(* Schneider Machine Expert - Basic project XNOR Gate, file version 2.9.0.0 *)
(* ProjectInformations: Name=New project *)

HARDWARE
  Cpu 0: TM221C24R
  EthernetConfiguration: NetworkName=M221, IpAllocationMode=FixedAddress, IpAddress=0.0.0.0, SubnetMask=0.0.0.0
  SerialLineConfiguration: Baud=Baud19200, Parity=ParityEven, DataBits=DataBits8, StopBits=StopBits1, PhysicalMedium=PhysicalMediumRs485, SlaveId=1, Addressing=SlaveAddressing
  MastTask: UsePeriodScanMode=false, PeriodScan=100
  FastTask: Period=255
  CpuBehavior: StartingMode=StartAsPreviousState, AutoSaveRamOnEeprom=true, WatchdogPeriod=250

SYMBOLS  (address, symbol, comment, settings)
  %I0.0     SWITCH_1
  %I0.1     SWITCH_2
  %Q0.0     MOTOR

POU New POU
  (* SectionNumber=1 *)

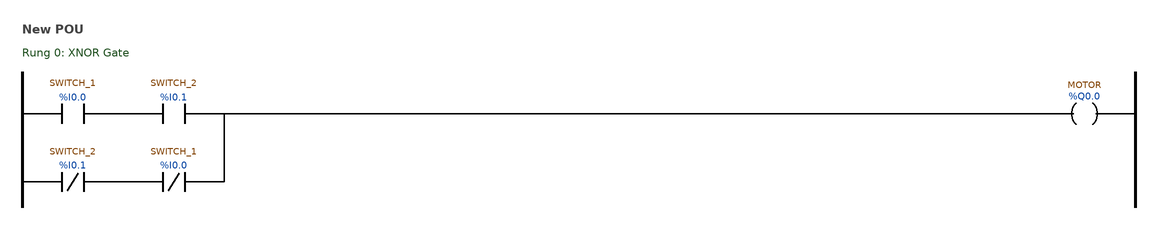

// Rung 0: XNOR Gate
  LD %I0.0                (* SWITCH_1 *)
  AND %I0.1               (* SWITCH_2 *)
  OR(N %I0.1              (* SWITCH_2 *)
  ANDN %I0.0              (* SWITCH_1 *)
  )
  ST %Q0.0                (* MOTOR *)
  // as ST:
  //   MOTOR := SWITCH_1 AND SWITCH_2 OR NOT SWITCH_2 AND NOT SWITCH_1;
